FUNCTION_BLOCK EL3351
VAR
	_io : EL3351_Data;
	{attribute addProperty Name "WcState"}
	_wcState : WcStateInputToggle;
	{attribute addProperty Name "Info data"}
	_infoData : InfoDataAds;
END_VAR

PROPERTY IO : REFERENCE TO EL3351_Data
GET
IO REF= _io;
END_GET
END_PROPERTY

PROPERTY WcState : REFERENCE TO WcStateInputToggle
GET
WcState REF= _wcState;
END_GET
END_PROPERTY

END_FUNCTION_BLOCK

(* stored: Version 1.1.0.1, ProductVersion 3.1.4024.9
   POU EL3351: Id {9fbde4d7-68ae-00a0-362e-bf4115f532f9}, SpecialFunc None
   Property IO: Id {f2a8869f-2f86-0c5a-0418-566701a5bbfb}
   Get Get: Id {959fe8d6-04cc-0dee-26f5-fd7d38672bfd}
   Property WcState: Id {1377d8cd-bd8f-0e10-2526-a5230a9d533f}
   Get Get: Id {61625ac2-c894-0e76-2b4b-f3bf61fd558c} *)
